TYPE ST_PROG_ENTRY :
STRUCT
  nMoverIndex     : UINT;
  MoveData        : ST_MOVE_DATA;
END_STRUCT
END_TYPE

(* stored: Version 1.1.0.1, ProductVersion 3.1.4024.15
   DUT ST_PROG_ENTRY: Id {fd9b93b6-3fa0-4c6c-a06c-d59d5361877e} *)
